RoboDK station: robot_station7x7.rdk

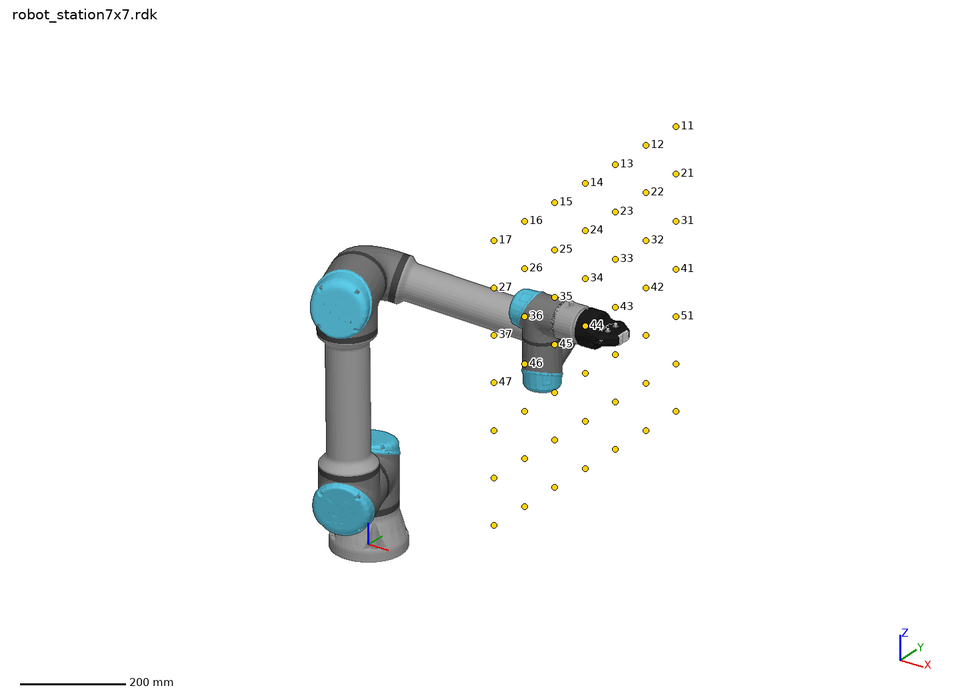
[picture v0: the station drawn from its stored meshes, robots at their saved joint values, targets as dots, program paths as lines]
Station test2. Poses are relative to the parent item; angles as X-Y-Z fixed-axis rotations.
  - frame UR5e Base at (0, 0, 0) mm
    - robot UR5e: 6 axes, payload 5 kg, reach 850 mm, repeatability 0.03 mm, weight 18.4 kg
        modified DH rows (alpha deg, a mm, theta deg, d mm): 0, 0, 0, 162.5; 90, 0, 180, 0; 0, 425, 0, 0; 0, 392.25, 0, 133.3; -90, 0, 0, 99.7; 90, 0, 180, 99.6
        joint limits [-360, -360, -360, -360, -360, -360] to [360, 360, 360, 360, 360, 360]; home [0, -90, -90, 0, 90, 0]; saved at [19.446, -89.342, -103.498, 12.84, 70.554, 0]
      - robot RobotiQ 2F85: 1 axes, payload 5 kg
          joint limits [0] to [85]; home [85]; saved at [85]
    - target 11 (Cartesian target) at (500, 300, 900) mm, rotated rx -90 ry 0 rz -90 deg; joints [63.261, -100.629, -45.238, -34.132, 26.739, 0] of UR5e
    - target 12 (Cartesian target) at (500, 200, 900) mm, rotated rx -90 ry 0 rz -90 deg; joints [55.331, -90.793, -56.345, -32.862, 34.669, 0] of UR5e
    - target 13 (Cartesian target) at (500, 100, 900) mm, rotated rx -90 ry 0 rz -90 deg; joints [43.311, -84.459, -62.341, -33.201, 46.689, 0] of UR5e
    - target 14 (Cartesian target) at (500, 0, 900) mm, rotated rx -90 ry 0 rz -90 deg; joints [26.343, -82.193, -64.264, -33.542, 63.657, 0] of UR5e
    - target 15 (Cartesian target) at (500, -100, 900) mm, rotated rx -90 ry 0 rz -90 deg; joints [6.487, -84.459, -62.341, -33.201, 83.513, 0] of UR5e
    - target 16 (Cartesian target) at (500, -200, 900) mm, rotated rx -90 ry 0 rz -90 deg; joints [-11.978, -90.793, -56.345, -32.862, 101.978, 0] of UR5e
    - target 17 (Cartesian target) at (500, -300, 900) mm, rotated rx -90 ry 0 rz -90 deg; joints [-26.662, -100.629, -45.238, -34.132, 116.663, 0] of UR5e
    - target 21 (Cartesian target) at (500, 300, 800) mm, rotated rx -90 ry 0 rz -90 deg; joints [63.261, -93.733, -69.417, -16.85, 26.739, 0] of UR5e
    - target 22 (Cartesian target) at (500, 200, 800) mm, rotated rx -90 ry 0 rz -90 deg; joints [55.331, -84.633, -78.37, -16.997, 34.669, 0] of UR5e
    - target 23 (Cartesian target) at (500, 100, 800) mm, rotated rx -90 ry 0 rz -90 deg; joints [43.311, -78.358, -83.591, -18.051, 46.689, 0] of UR5e
    - target 24 (Cartesian target) at (500, 0, 800) mm, rotated rx -90 ry 0 rz -90 deg; joints [26.343, -76.047, -85.318, -18.635, 63.657, 0] of UR5e
    - target 25 (Cartesian target) at (500, -100, 800) mm, rotated rx -90 ry 0 rz -90 deg; joints [6.487, -78.358, -83.591, -18.051, 83.513, 0] of UR5e
    - target 26 (Cartesian target) at (500, -200, 800) mm, rotated rx -90 ry 0 rz -90 deg; joints [-11.978, -84.633, -78.37, -16.997, 101.978, 0] of UR5e
    - target 27 (Cartesian target) at (500, -300, 800) mm, rotated rx -90 ry 0 rz -90 deg; joints [-26.662, -93.733, -69.417, -16.85, 116.663, 0] of UR5e
    - target 31 (Cartesian target) at (500, 300, 700) mm, rotated rx -90 ry 0 rz -90 deg; joints [63.261, -91.489, -86.62, -1.891, 26.739, 0] of UR5e
    - target 32 (Cartesian target) at (500, 200, 700) mm, rotated rx -90 ry 0 rz -90 deg; joints [55.331, -82.356, -95.222, -2.422, 34.669, 0] of UR5e
    - target 33 (Cartesian target) at (500, 100, 700) mm, rotated rx -90 ry 0 rz -90 deg; joints [43.311, -75.804, -100.428, -3.768, 46.689, 0] of UR5e
    - target 34 (Cartesian target) at (500, 0, 700) mm, rotated rx -90 ry 0 rz -90 deg; joints [26.343, -73.34, -102.18, -4.48, 63.657, 0] of UR5e
    - target 35 (Cartesian target) at (500, -100, 700) mm, rotated rx -90 ry 0 rz -90 deg; joints [6.487, -75.804, -100.428, -3.768, 83.513, 0] of UR5e
    - target 36 (Cartesian target) at (500, -200, 700) mm, rotated rx -90 ry 0 rz -90 deg; joints [-11.978, -82.356, -95.222, -2.422, 101.978, 0] of UR5e
    - target 37 (Cartesian target) at (500, -300, 700) mm, rotated rx -90 ry 0 rz -90 deg; joints [-26.662, -91.489, -86.62, -1.891, 116.663, 0] of UR5e
    - target 41 (Cartesian target) at (500, 300, 600) mm, rotated rx -90 ry 0 rz -90 deg; joints [63.261, -92.769, -100.001, 12.77, 26.739, 0] of UR5e
    - target 42 (Cartesian target) at (500, 200, 600) mm, rotated rx -90 ry 0 rz -90 deg; joints [55.331, -83.56, -108.883, 12.443, 34.669, 0] of UR5e
    - target 43 (Cartesian target) at (500, 100, 600) mm, rotated rx -90 ry 0 rz -90 deg; joints [43.311, -76.714, -114.432, 11.146, 46.689, 0] of UR5e
    - target 44 (Cartesian target) at (500, 0, 600) mm, rotated rx -90 ry 0 rz -90 deg; joints [26.343, -74.079, -116.334, 10.413, 63.657, 0] of UR5e
    - target 45 (Cartesian target) at (500, -100, 600) mm, rotated rx -90 ry 0 rz -90 deg; joints [6.487, -76.714, -114.432, 11.146, 83.513, 0] of UR5e
    - target 46 (Cartesian target) at (500, -200, 600) mm, rotated rx -90 ry 0 rz -90 deg; joints [-11.978, -83.56, -108.883, 12.443, 101.978, 0] of UR5e
    - target 47 (Cartesian target) at (500, -300, 600) mm, rotated rx -90 ry 0 rz -90 deg; joints [-26.662, -92.769, -100.001, 12.77, 116.663, 0] of UR5e
    - target 51 (Cartesian target) at (500, 300, 500) mm, rotated rx -90 ry 0 rz -90 deg; joints [63.261, -97.622, -110.262, 27.884, 26.739, 0] of UR5e
    - target 52 (Cartesian target) at (500, 200, 500) mm, rotated rx -90 ry 0 rz -90 deg; joints [55.331, -88.735, -119.754, 28.489, 34.669, 0] of UR5e
    - target 53 (Cartesian target) at (500, 100, 500) mm, rotated rx -90 ry 0 rz -90 deg; joints [43.311, -81.914, -125.892, 27.806, 46.689, 0] of UR5e
    - target 54 (Cartesian target) at (500, 0, 500) mm, rotated rx -90 ry 0 rz -90 deg; joints [26.343, -79.225, -128.043, 27.267, 63.657, 0] of UR5e
    - target 55 (Cartesian target) at (500, -100, 500) mm, rotated rx -90 ry 0 rz -90 deg; joints [6.487, -81.914, -125.892, 27.806, 83.513, 0] of UR5e
    - target 56 (Cartesian target) at (500, -200, 500) mm, rotated rx -90 ry 0 rz -90 deg; joints [-11.978, -88.735, -119.754, 28.489, 101.978, 0] of UR5e
    - target 57 (Cartesian target) at (500, -300, 500) mm, rotated rx -90 ry 0 rz -90 deg; joints [-26.662, -97.622, -110.262, 27.884, 116.663, 0] of UR5e
    - target 61 (Cartesian target) at (500, 300, 400) mm, rotated rx -90 ry 0 rz -90 deg; joints [63.261, -106.231, -117.32, 43.551, 26.739, 0] of UR5e
    - target 62 (Cartesian target) at (500, 200, 400) mm, rotated rx -90 ry 0 rz -90 deg; joints [55.331, -98.553, -127.512, 46.066, 34.669, 0] of UR5e
    - target 63 (Cartesian target) at (500, 100, 400) mm, rotated rx -90 ry 0 rz -90 deg; joints [43.311, -92.634, -134.34, 46.974, 46.689, 0] of UR5e
    - target 64 (Cartesian target) at (500, 0, 400) mm, rotated rx -90 ry 0 rz -90 deg; joints [26.343, -90.275, -136.794, 47.069, 63.657, 0] of UR5e
    - target 65 (Cartesian target) at (500, -100, 400) mm, rotated rx -90 ry 0 rz -90 deg; joints [6.487, -92.634, -134.34, 46.974, 83.513, 0] of UR5e
    - target 66 (Cartesian target) at (500, -200, 400) mm, rotated rx -90 ry 0 rz -90 deg; joints [-11.978, -98.553, -127.512, 46.066, 101.978, 0] of UR5e
    - target 67 (Cartesian target) at (500, -300, 400) mm, rotated rx -90 ry 0 rz -90 deg; joints [-26.662, -106.231, -117.32, 43.551, 116.663, 0] of UR5e
    - target 71 (Cartesian target) at (500, 300, 300) mm, rotated rx -90 ry 0 rz -90 deg; joints [63.261, -118.289, -120.773, 59.062, 26.739, 0] of UR5e
    - target 72 (Cartesian target) at (500, 200, 300) mm, rotated rx -90 ry 0 rz -90 deg; joints [55.331, -112.933, -131.422, 64.355, 34.669, 0] of UR5e
    - target 73 (Cartesian target) at (500, 100, 300) mm, rotated rx -90 ry 0 rz -90 deg; joints [43.311, -109.212, -138.727, 67.939, 46.689, 0] of UR5e
    - target 74 (Cartesian target) at (500, 0, 300) mm, rotated rx -90 ry 0 rz -90 deg; joints [26.343, -107.834, -141.404, 69.238, 63.657, 0] of UR5e
    - target 75 (Cartesian target) at (500, -100, 300) mm, rotated rx -90 ry 0 rz -90 deg; joints [6.487, -109.212, -138.727, 67.939, 83.513, 0] of UR5e
    - target 76 (Cartesian target) at (500, -200, 300) mm, rotated rx -90 ry 0 rz -90 deg; joints [-11.978, -112.933, -131.422, 64.355, 101.978, 0] of UR5e
    - target 77 (Cartesian target) at (500, -300, 300) mm, rotated rx -90 ry 0 rz -90 deg; joints [-26.662, -118.289, -120.773, 59.062, 116.663, 0] of UR5e
